Fanuc KAREL source: compact_preamble.KL

PROGRAM KA00144
%NOLOCKGROUP
VAR
SRC : ARRAY[2] OF SHORT
DST : ARRAY[2] OF SHORT
BEGIN
SRC[1]=2
DST[1]=SRC[1]
END KA00144
